// TIA Portal V20 export
TYPE "LER_typeRFIDConfiguration"
// stored: Access Published
   STRUCT
      referenceDesignator : WString[25];
      addrTag : DWord;
      lengthData : Word := 16#100;
      attribute : Byte := 16#81;
      duration : Word := 16#1;
      durUnit : Word := 16#2;
   END_STRUCT;
END_TYPE
